TYPE "udtModbusValBool"
VERSION : 0.1
   STRUCT
      iAddr { ExternalAccessible := 'False'; ExternalVisible := 'False'; ExternalWritable := 'False'} : UInt;   // Full modbus address (1 indexed, including offset for object type)
      bVal { ExternalAccessible := 'False'; ExternalVisible := 'False'; ExternalWritable := 'False'} : Bool;
   END_STRUCT;

END_TYPE

